// TIA Portal V20 export
DATA_BLOCK "InstLimitValueDataset1"   // DB54
TITLE = Instanz LimitValueDataset1 / Instance LimitValueDataset1
{ DB_Accessible_From_OPC_UA := 'FALSE' }
AUTHOR : SICAR
FAMILY : ProdData
// Instanz DB / Instance DB
// stored: DBAccessibleFromOPCUA false, InstanceOfName LSicar_ProdDataLimitValues, InstanceOfType FB
"LSicar_ProdDataLimitValues"
   // VAR_INPUT
   //    numberConfigDataSets { ExternalAccessible := 'False'; ExternalVisible := 'False'; ExternalWritable := 'False'} : Int := 0;
   //    dataSetNumber { ExternalAccessible := 'False'; ExternalVisible := 'False'; ExternalWritable := 'False'} : UInt := 0;
   // END_VAR
   // VAR_IN_OUT
   //    numberOfDataSets : "LSicar_typeNumberOfDataSets";
   //    dataSet : "LSicar_typeLimitValue";
   //    colorCodeSelectButton { ExternalAccessible := 'False'; ExternalVisible := 'False'; ExternalWritable := 'False'} : UInt := 0;
   // END_VAR
   // VAR
   //    statLimitValue { ExternalAccessible := 'False'; ExternalVisible := 'False'; ExternalWritable := 'False'} : Array[0..10] of "LSicar_typeEdgePulseStruct";
   //    statPrewarnActive { ExternalAccessible := 'False'; ExternalVisible := 'False'; ExternalWritable := 'False'} : Bool := FALSE;
   //    statAlarmActive { ExternalAccessible := 'False'; ExternalVisible := 'False'; ExternalWritable := 'False'} : Bool := FALSE;
   // END_VAR
BEGIN
   statLimitValue[0..10].risEdgeCountUp := FALSE;
   statLimitValue[0..10].posPulseCountUp := FALSE;
   statLimitValue[0..10].risEdgeCountDown := FALSE;
   statLimitValue[0..10].posPulseCountDown := FALSE;
   statLimitValue[0..10].risEdgeReset := FALSE;
   statLimitValue[0..10].posPulseReset := FALSE;
END_DATA_BLOCK
